// TIA Portal V17 export
// export: Created 2025-03-05T07:59:45.6753335Z, ExportSetting WithDefaults, DisplayName Totally Integrated Automation Portal, DisplayVersion V17 Update 8, DisplayName TIA Portal Openness, DisplayVersion V17 Update 8, DisplayName TIA Portal Version Control Interface, DisplayVersion V17, DisplayName SINAMICS Startdrive Advanced, DisplayVersion V17 SP2, DisplayName SINAMICS Startdrive G110M, G120, G120C, G120D, G120P, G115D, DisplayVersion V17 SP2, DisplayName SINAMICS Startdrive G130, G150, S120, S150, SINAMICS MV, S210, DisplayVersion V17 SP2, DisplayName STEP 7 Professional, DisplayVersion V17 Update 8, DisplayName SINUMERIK ONE STEP 7 Toolbox, DisplayVersion V17 Update 12, DisplayName SINUMERIK 840D sl STEP 7 Toolbox, DisplayVersion V17 Update 12, DisplayName STEP 7 Safety, DisplayVersion V17 Update 6, DisplayName WinCC Advanced, DisplayVersion V17 Update 8
FUNCTION "FC326_CHANNEL_6" : Void   // FC326, LAD
{ S7_Optimized_Access := 'FALSE' }
AUTHOR : ETXETAR
VERSION : 1.0
// stored: AutoNumber false, IsIECCheckEnabled false, SetENOAutomatically false, UDAEnableTagReadback false
   VAR_TEMP
      NC_RESET_CH2 : Bool;
      NC_START_CH2 : Bool;
   END_VAR
BEGIN

REGION Network 1: RESET CHANNEL
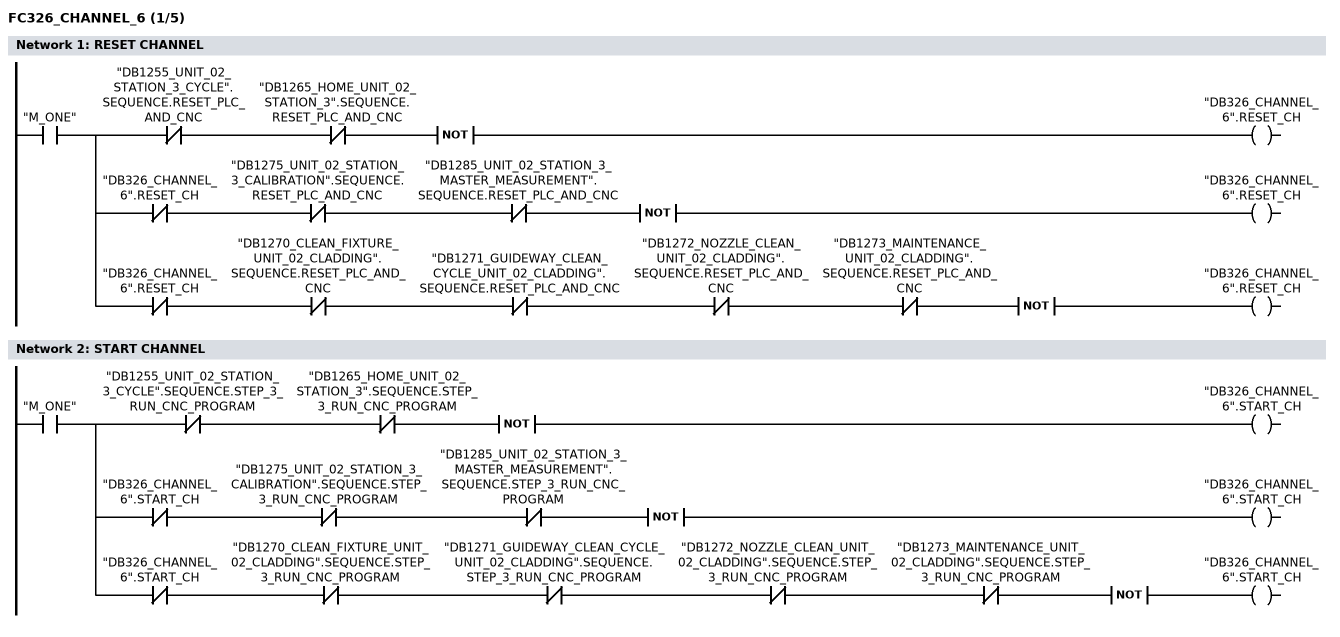
   RUNG wire#powerrail
      Contact( "M_ONE" )
      wire#w1
      I_Contact( "DB1255_UNIT_02_STATION_3_CYCLE".SEQUENCE.RESET_PLC_AND_CNC )
      I_Contact( "DB1265_HOME_UNIT_02_STATION_3".SEQUENCE.RESET_PLC_AND_CNC )
      Not()
      Coil( "DB326_CHANNEL_6".RESET_CH )
   END_RUNG
   RUNG wire#w1
      I_Contact( "DB326_CHANNEL_6".RESET_CH )
      I_Contact( "DB1275_UNIT_02_STATION_3_CALIBRATION".SEQUENCE.RESET_PLC_AND_CNC )
      I_Contact( "DB1285_UNIT_02_STATION_3_MASTER_MEASUREMENT".SEQUENCE.RESET_PLC_AND_CNC )
      Not()
      Coil( "DB326_CHANNEL_6".RESET_CH )
   END_RUNG
   RUNG wire#w1
      I_Contact( "DB326_CHANNEL_6".RESET_CH )
      I_Contact( "DB1270_CLEAN_FIXTURE_UNIT_02_CLADDING".SEQUENCE.RESET_PLC_AND_CNC )
      I_Contact( "DB1271_GUIDEWAY_CLEAN_CYCLE_UNIT_02_CLADDING".SEQUENCE.RESET_PLC_AND_CNC )
      I_Contact( "DB1272_NOZZLE_CLEAN_UNIT_02_CLADDING".SEQUENCE.RESET_PLC_AND_CNC )
      I_Contact( "DB1273_MAINTENANCE_UNIT_02_CLADDING".SEQUENCE.RESET_PLC_AND_CNC )
      Not()
      Coil( "DB326_CHANNEL_6".RESET_CH )
   END_RUNG
   // the same network as SCL:
   "DB326_CHANNEL_6".RESET_CH := NOT ("M_ONE" AND NOT "DB1255_UNIT_02_STATION_3_CYCLE".SEQUENCE.RESET_PLC_AND_CNC AND NOT "DB1265_HOME_UNIT_02_STATION_3".SEQUENCE.RESET_PLC_AND_CNC);
   "DB326_CHANNEL_6".RESET_CH := NOT ("M_ONE" AND NOT "DB326_CHANNEL_6".RESET_CH AND NOT "DB1275_UNIT_02_STATION_3_CALIBRATION".SEQUENCE.RESET_PLC_AND_CNC AND NOT "DB1285_UNIT_02_STATION_3_MASTER_MEASUREMENT".SEQUENCE.RESET_PLC_AND_CNC);
   "DB326_CHANNEL_6".RESET_CH := NOT ("M_ONE" AND NOT "DB326_CHANNEL_6".RESET_CH AND NOT "DB1270_CLEAN_FIXTURE_UNIT_02_CLADDING".SEQUENCE.RESET_PLC_AND_CNC AND NOT "DB1271_GUIDEWAY_CLEAN_CYCLE_UNIT_02_CLADDING".SEQUENCE.RESET_PLC_AND_CNC AND NOT "DB1272_NOZZLE_CLEAN_UNIT_02_CLADDING".SEQUENCE.RESET_PLC_AND_CNC AND NOT "DB1273_MAINTENANCE_UNIT_02_CLADDING".SEQUENCE.RESET_PLC_AND_CNC);
END_REGION

REGION Network 2: START CHANNEL
   RUNG wire#powerrail
      Contact( "M_ONE" )
      wire#w1
      I_Contact( "DB1255_UNIT_02_STATION_3_CYCLE".SEQUENCE.STEP_3_RUN_CNC_PROGRAM )
      I_Contact( "DB1265_HOME_UNIT_02_STATION_3".SEQUENCE.STEP_3_RUN_CNC_PROGRAM )
      Not()
      Coil( "DB326_CHANNEL_6".START_CH )
   END_RUNG
   RUNG wire#w1
      I_Contact( "DB326_CHANNEL_6".START_CH )
      I_Contact( "DB1275_UNIT_02_STATION_3_CALIBRATION".SEQUENCE.STEP_3_RUN_CNC_PROGRAM )
      I_Contact( "DB1285_UNIT_02_STATION_3_MASTER_MEASUREMENT".SEQUENCE.STEP_3_RUN_CNC_PROGRAM )
      Not()
      Coil( "DB326_CHANNEL_6".START_CH )
   END_RUNG
   RUNG wire#w1
      I_Contact( "DB326_CHANNEL_6".START_CH )
      I_Contact( "DB1270_CLEAN_FIXTURE_UNIT_02_CLADDING".SEQUENCE.STEP_3_RUN_CNC_PROGRAM )
      I_Contact( "DB1271_GUIDEWAY_CLEAN_CYCLE_UNIT_02_CLADDING".SEQUENCE.STEP_3_RUN_CNC_PROGRAM )
      I_Contact( "DB1272_NOZZLE_CLEAN_UNIT_02_CLADDING".SEQUENCE.STEP_3_RUN_CNC_PROGRAM )
      I_Contact( "DB1273_MAINTENANCE_UNIT_02_CLADDING".SEQUENCE.STEP_3_RUN_CNC_PROGRAM )
      Not()
      Coil( "DB326_CHANNEL_6".START_CH )
   END_RUNG
   // the same network as SCL:
   "DB326_CHANNEL_6".START_CH := NOT ("M_ONE" AND NOT "DB1255_UNIT_02_STATION_3_CYCLE".SEQUENCE.STEP_3_RUN_CNC_PROGRAM AND NOT "DB1265_HOME_UNIT_02_STATION_3".SEQUENCE.STEP_3_RUN_CNC_PROGRAM);
   "DB326_CHANNEL_6".START_CH := NOT ("M_ONE" AND NOT "DB326_CHANNEL_6".START_CH AND NOT "DB1275_UNIT_02_STATION_3_CALIBRATION".SEQUENCE.STEP_3_RUN_CNC_PROGRAM AND NOT "DB1285_UNIT_02_STATION_3_MASTER_MEASUREMENT".SEQUENCE.STEP_3_RUN_CNC_PROGRAM);
   "DB326_CHANNEL_6".START_CH := NOT ("M_ONE" AND NOT "DB326_CHANNEL_6".START_CH AND NOT "DB1270_CLEAN_FIXTURE_UNIT_02_CLADDING".SEQUENCE.STEP_3_RUN_CNC_PROGRAM AND NOT "DB1271_GUIDEWAY_CLEAN_CYCLE_UNIT_02_CLADDING".SEQUENCE.STEP_3_RUN_CNC_PROGRAM AND NOT "DB1272_NOZZLE_CLEAN_UNIT_02_CLADDING".SEQUENCE.STEP_3_RUN_CNC_PROGRAM AND NOT "DB1273_MAINTENANCE_UNIT_02_CLADDING".SEQUENCE.STEP_3_RUN_CNC_PROGRAM);
END_REGION

REGION Network 3: CALL FB321 CHANNEL 6 / CHANNEL 3 XFLEX-DUO
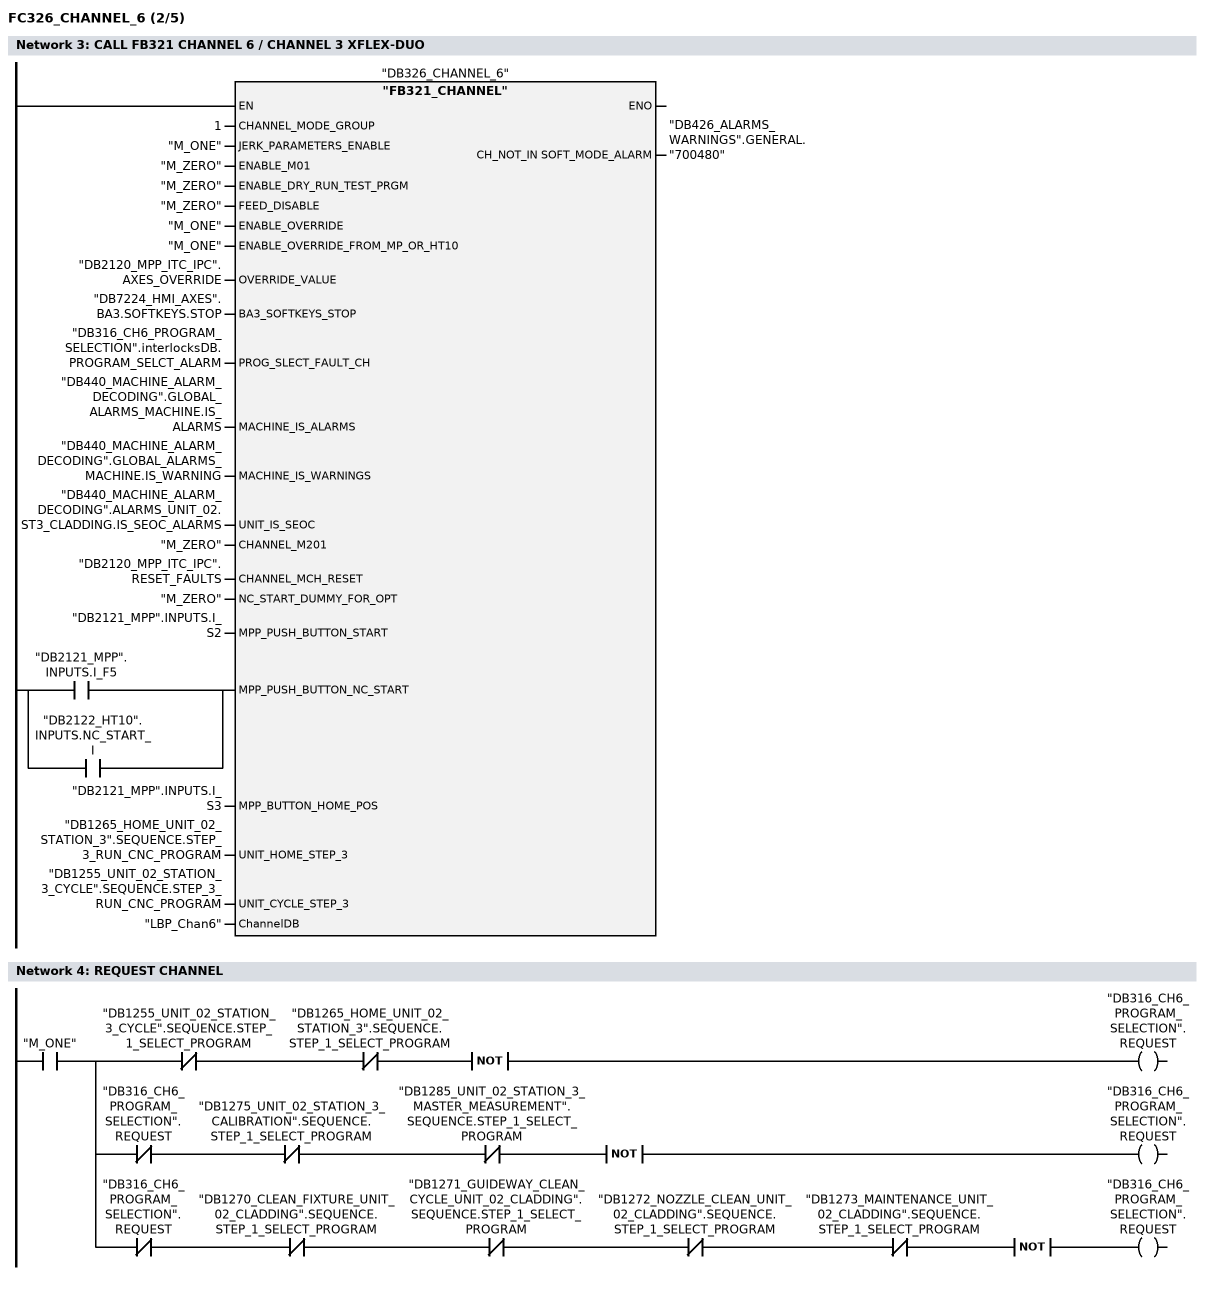
   RUNG wire#powerrail
      "DB326_CHANNEL_6"(MPP_PUSH_BUTTON_NC_START := wire#w1, CHANNEL_MODE_GROUP := 1, JERK_PARAMETERS_ENABLE := "M_ONE", ENABLE_M01 := "M_ZERO", ENABLE_DRY_RUN_TEST_PRGM := "M_ZERO", FEED_DISABLE := "M_ZERO", ENABLE_OVERRIDE := "M_ONE", ENABLE_OVERRIDE_FROM_MP_OR_HT10 := "M_ONE", OVERRIDE_VALUE := "DB2120_MPP_ITC_IPC".AXES_OVERRIDE, BA3_SOFTKEYS_STOP := "DB7224_HMI_AXES".BA3.SOFTKEYS.STOP, PROG_SLECT_FAULT_CH := "DB316_CH6_PROGRAM_SELECTION".interlocksDB.PROGRAM_SELCT_ALARM, MACHINE_IS_ALARMS := "DB440_MACHINE_ALARM_DECODING".GLOBAL_ALARMS_MACHINE.IS_ALARMS, MACHINE_IS_WARNINGS := "DB440_MACHINE_ALARM_DECODING".GLOBAL_ALARMS_MACHINE.IS_WARNING, UNIT_IS_SEOC := "DB440_MACHINE_ALARM_DECODING".ALARMS_UNIT_02.ST3_CLADDING.IS_SEOC_ALARMS, CHANNEL_M201 := "M_ZERO", CHANNEL_MCH_RESET := "DB2120_MPP_ITC_IPC".RESET_FAULTS, NC_START_DUMMY_FOR_OPT := "M_ZERO", MPP_PUSH_BUTTON_START := "DB2121_MPP".INPUTS.I_S2, MPP_BUTTON_HOME_POS := "DB2121_MPP".INPUTS.I_S3, UNIT_HOME_STEP_3 := "DB1265_HOME_UNIT_02_STATION_3".SEQUENCE.STEP_3_RUN_CNC_PROGRAM, UNIT_CYCLE_STEP_3 := "DB1255_UNIT_02_STATION_3_CYCLE".SEQUENCE.STEP_3_RUN_CNC_PROGRAM, ChannelDB := "LBP_Chan6", "CH_NOT_IN SOFT_MODE_ALARM" => "DB426_ALARMS_WARNINGS".GENERAL."700480")
   END_RUNG
   RUNG wire#powerrail
      Contact( "DB2121_MPP".INPUTS.I_F5 )
   END_RUNG wire#w1
   RUNG wire#powerrail
      Contact( "DB2122_HT10".INPUTS.NC_START_I )
   END_RUNG wire#w1
   // the same network as SCL:
   "DB326_CHANNEL_6"(CHANNEL_MODE_GROUP := 1,   // "FB321_CHANNEL"
                     JERK_PARAMETERS_ENABLE := "M_ONE",
                     ENABLE_M01 := "M_ZERO",
                     ENABLE_DRY_RUN_TEST_PRGM := "M_ZERO",
                     FEED_DISABLE := "M_ZERO",
                     ENABLE_OVERRIDE := "M_ONE",
                     ENABLE_OVERRIDE_FROM_MP_OR_HT10 := "M_ONE",
                     OVERRIDE_VALUE := "DB2120_MPP_ITC_IPC".AXES_OVERRIDE,
                     BA3_SOFTKEYS_STOP := "DB7224_HMI_AXES".BA3.SOFTKEYS.STOP,
                     PROG_SLECT_FAULT_CH := "DB316_CH6_PROGRAM_SELECTION".interlocksDB.PROGRAM_SELCT_ALARM,
                     MACHINE_IS_ALARMS := "DB440_MACHINE_ALARM_DECODING".GLOBAL_ALARMS_MACHINE.IS_ALARMS,
                     MACHINE_IS_WARNINGS := "DB440_MACHINE_ALARM_DECODING".GLOBAL_ALARMS_MACHINE.IS_WARNING,
                     UNIT_IS_SEOC := "DB440_MACHINE_ALARM_DECODING".ALARMS_UNIT_02.ST3_CLADDING.IS_SEOC_ALARMS,
                     CHANNEL_M201 := "M_ZERO",
                     CHANNEL_MCH_RESET := "DB2120_MPP_ITC_IPC".RESET_FAULTS,
                     NC_START_DUMMY_FOR_OPT := "M_ZERO",
                     MPP_PUSH_BUTTON_START := "DB2121_MPP".INPUTS.I_S2,
                     MPP_PUSH_BUTTON_NC_START := "DB2121_MPP".INPUTS.I_F5 OR "DB2122_HT10".INPUTS.NC_START_I,
                     MPP_BUTTON_HOME_POS := "DB2121_MPP".INPUTS.I_S3,
                     UNIT_HOME_STEP_3 := "DB1265_HOME_UNIT_02_STATION_3".SEQUENCE.STEP_3_RUN_CNC_PROGRAM,
                     UNIT_CYCLE_STEP_3 := "DB1255_UNIT_02_STATION_3_CYCLE".SEQUENCE.STEP_3_RUN_CNC_PROGRAM,
                     ChannelDB := "LBP_Chan6",
                     "CH_NOT_IN SOFT_MODE_ALARM" => "DB426_ALARMS_WARNINGS".GENERAL."700480");
END_REGION

REGION Network 4: REQUEST CHANNEL
   RUNG wire#powerrail
      Contact( "M_ONE" )
      wire#w1
      I_Contact( "DB1255_UNIT_02_STATION_3_CYCLE".SEQUENCE.STEP_1_SELECT_PROGRAM )
      I_Contact( "DB1265_HOME_UNIT_02_STATION_3".SEQUENCE.STEP_1_SELECT_PROGRAM )
      Not()
      Coil( "DB316_CH6_PROGRAM_SELECTION".REQUEST )
   END_RUNG
   RUNG wire#w1
      I_Contact( "DB316_CH6_PROGRAM_SELECTION".REQUEST )
      I_Contact( "DB1275_UNIT_02_STATION_3_CALIBRATION".SEQUENCE.STEP_1_SELECT_PROGRAM )
      I_Contact( "DB1285_UNIT_02_STATION_3_MASTER_MEASUREMENT".SEQUENCE.STEP_1_SELECT_PROGRAM )
      Not()
      Coil( "DB316_CH6_PROGRAM_SELECTION".REQUEST )
   END_RUNG
   RUNG wire#w1
      I_Contact( "DB316_CH6_PROGRAM_SELECTION".REQUEST )
      I_Contact( "DB1270_CLEAN_FIXTURE_UNIT_02_CLADDING".SEQUENCE.STEP_1_SELECT_PROGRAM )
      I_Contact( "DB1271_GUIDEWAY_CLEAN_CYCLE_UNIT_02_CLADDING".SEQUENCE.STEP_1_SELECT_PROGRAM )
      I_Contact( "DB1272_NOZZLE_CLEAN_UNIT_02_CLADDING".SEQUENCE.STEP_1_SELECT_PROGRAM )
      I_Contact( "DB1273_MAINTENANCE_UNIT_02_CLADDING".SEQUENCE.STEP_1_SELECT_PROGRAM )
      Not()
      Coil( "DB316_CH6_PROGRAM_SELECTION".REQUEST )
   END_RUNG
   // the same network as SCL:
   "DB316_CH6_PROGRAM_SELECTION".REQUEST := NOT ("M_ONE" AND NOT "DB1255_UNIT_02_STATION_3_CYCLE".SEQUENCE.STEP_1_SELECT_PROGRAM AND NOT "DB1265_HOME_UNIT_02_STATION_3".SEQUENCE.STEP_1_SELECT_PROGRAM);
   "DB316_CH6_PROGRAM_SELECTION".REQUEST := NOT ("M_ONE" AND NOT "DB316_CH6_PROGRAM_SELECTION".REQUEST AND NOT "DB1275_UNIT_02_STATION_3_CALIBRATION".SEQUENCE.STEP_1_SELECT_PROGRAM AND NOT "DB1285_UNIT_02_STATION_3_MASTER_MEASUREMENT".SEQUENCE.STEP_1_SELECT_PROGRAM);
   "DB316_CH6_PROGRAM_SELECTION".REQUEST := NOT ("M_ONE" AND NOT "DB316_CH6_PROGRAM_SELECTION".REQUEST AND NOT "DB1270_CLEAN_FIXTURE_UNIT_02_CLADDING".SEQUENCE.STEP_1_SELECT_PROGRAM AND NOT "DB1271_GUIDEWAY_CLEAN_CYCLE_UNIT_02_CLADDING".SEQUENCE.STEP_1_SELECT_PROGRAM AND NOT "DB1272_NOZZLE_CLEAN_UNIT_02_CLADDING".SEQUENCE.STEP_1_SELECT_PROGRAM AND NOT "DB1273_MAINTENANCE_UNIT_02_CLADDING".SEQUENCE.STEP_1_SELECT_PROGRAM);
END_REGION

REGION Network 5: CALL FB311 CHANNEL PROGRAM SELECTION / CHANNEL 3 X-FLEX DUO
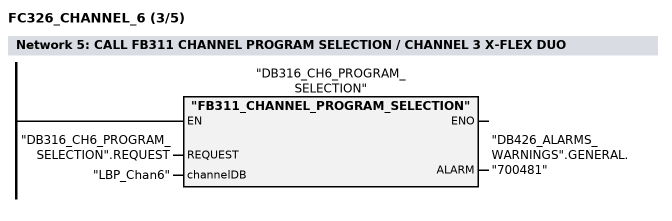
   RUNG wire#powerrail
      "DB316_CH6_PROGRAM_SELECTION"(REQUEST := "DB316_CH6_PROGRAM_SELECTION".REQUEST, channelDB := "LBP_Chan6", ALARM => "DB426_ALARMS_WARNINGS".GENERAL."700481")
   END_RUNG
   // the same network as SCL:
   "DB316_CH6_PROGRAM_SELECTION"(REQUEST := "DB316_CH6_PROGRAM_SELECTION".REQUEST,   // "FB311_CHANNEL_PROGRAM_SELECTION"
                           channelDB := "LBP_Chan6",
                           ALARM => "DB426_ALARMS_WARNINGS".GENERAL."700481");
END_REGION

REGION Network 6: CALL FB301 CHANNEL READ AXES POSITIONS
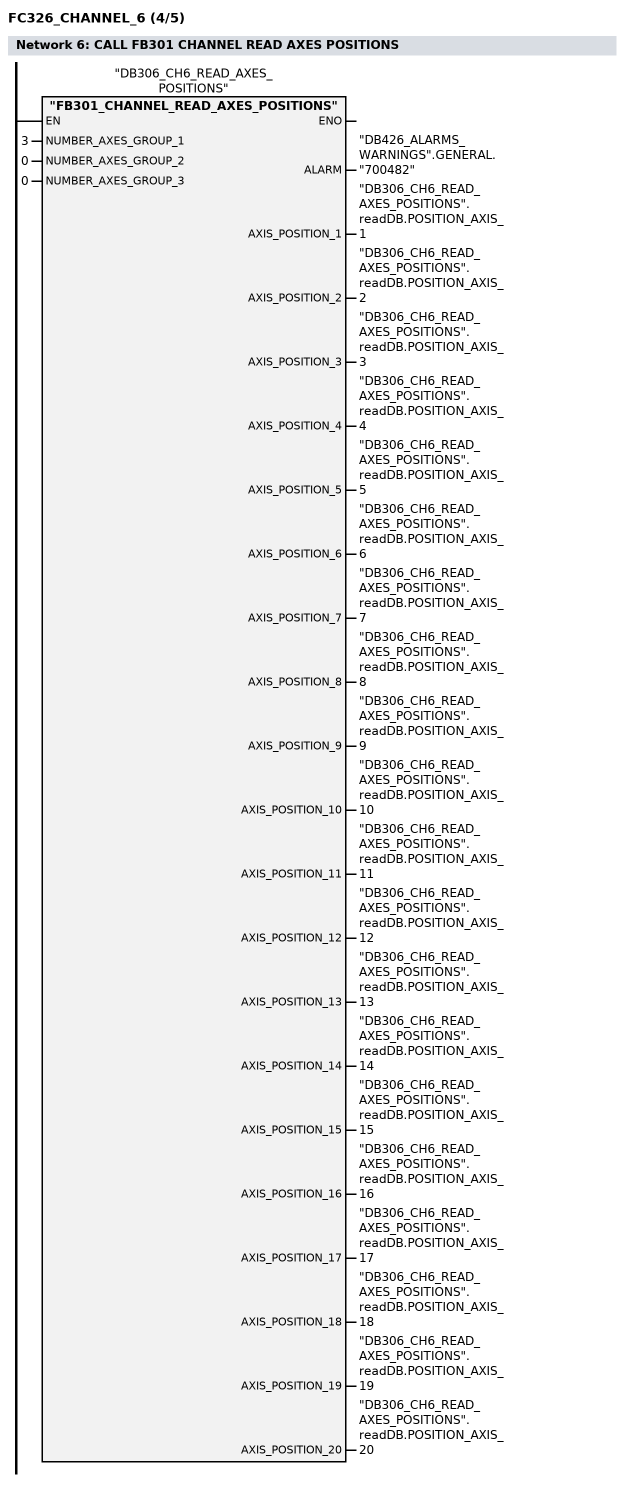
   RUNG wire#powerrail
      "DB306_CH6_READ_AXES_POSITIONS"(NUMBER_AXES_GROUP_1 := 3, NUMBER_AXES_GROUP_2 := 0, NUMBER_AXES_GROUP_3 := 0, ALARM => "DB426_ALARMS_WARNINGS".GENERAL."700482", AXIS_POSITION_1 => "DB306_CH6_READ_AXES_POSITIONS".readDB.POSITION_AXIS_1, AXIS_POSITION_2 => "DB306_CH6_READ_AXES_POSITIONS".readDB.POSITION_AXIS_2, AXIS_POSITION_3 => "DB306_CH6_READ_AXES_POSITIONS".readDB.POSITION_AXIS_3, AXIS_POSITION_4 => "DB306_CH6_READ_AXES_POSITIONS".readDB.POSITION_AXIS_4, AXIS_POSITION_5 => "DB306_CH6_READ_AXES_POSITIONS".readDB.POSITION_AXIS_5, AXIS_POSITION_6 => "DB306_CH6_READ_AXES_POSITIONS".readDB.POSITION_AXIS_6, AXIS_POSITION_7 => "DB306_CH6_READ_AXES_POSITIONS".readDB.POSITION_AXIS_7, AXIS_POSITION_8 => "DB306_CH6_READ_AXES_POSITIONS".readDB.POSITION_AXIS_8, AXIS_POSITION_9 => "DB306_CH6_READ_AXES_POSITIONS".readDB.POSITION_AXIS_9, AXIS_POSITION_10 => "DB306_CH6_READ_AXES_POSITIONS".readDB.POSITION_AXIS_10, AXIS_POSITION_11 => "DB306_CH6_READ_AXES_POSITIONS".readDB.POSITION_AXIS_11, AXIS_POSITION_12 => "DB306_CH6_READ_AXES_POSITIONS".readDB.POSITION_AXIS_12, AXIS_POSITION_13 => "DB306_CH6_READ_AXES_POSITIONS".readDB.POSITION_AXIS_13, AXIS_POSITION_14 => "DB306_CH6_READ_AXES_POSITIONS".readDB.POSITION_AXIS_14, AXIS_POSITION_15 => "DB306_CH6_READ_AXES_POSITIONS".readDB.POSITION_AXIS_15, AXIS_POSITION_16 => "DB306_CH6_READ_AXES_POSITIONS".readDB.POSITION_AXIS_16, AXIS_POSITION_17 => "DB306_CH6_READ_AXES_POSITIONS".readDB.POSITION_AXIS_17, AXIS_POSITION_18 => "DB306_CH6_READ_AXES_POSITIONS".readDB.POSITION_AXIS_18, AXIS_POSITION_19 => "DB306_CH6_READ_AXES_POSITIONS".readDB.POSITION_AXIS_19, AXIS_POSITION_20 => "DB306_CH6_READ_AXES_POSITIONS".readDB.POSITION_AXIS_20)
   END_RUNG
   // the same network as SCL:
   "DB306_CH6_READ_AXES_POSITIONS"(NUMBER_AXES_GROUP_1 := 3,   // "FB301_CHANNEL_READ_AXES_POSITIONS"
                           NUMBER_AXES_GROUP_2 := 0,
                           NUMBER_AXES_GROUP_3 := 0,
                           ALARM => "DB426_ALARMS_WARNINGS".GENERAL."700482",
                           AXIS_POSITION_1 => "DB306_CH6_READ_AXES_POSITIONS".readDB.POSITION_AXIS_1,
                           AXIS_POSITION_2 => "DB306_CH6_READ_AXES_POSITIONS".readDB.POSITION_AXIS_2,
                           AXIS_POSITION_3 => "DB306_CH6_READ_AXES_POSITIONS".readDB.POSITION_AXIS_3,
                           AXIS_POSITION_4 => "DB306_CH6_READ_AXES_POSITIONS".readDB.POSITION_AXIS_4,
                           AXIS_POSITION_5 => "DB306_CH6_READ_AXES_POSITIONS".readDB.POSITION_AXIS_5,
                           AXIS_POSITION_6 => "DB306_CH6_READ_AXES_POSITIONS".readDB.POSITION_AXIS_6,
                           AXIS_POSITION_7 => "DB306_CH6_READ_AXES_POSITIONS".readDB.POSITION_AXIS_7,
                           AXIS_POSITION_8 => "DB306_CH6_READ_AXES_POSITIONS".readDB.POSITION_AXIS_8,
                           AXIS_POSITION_9 => "DB306_CH6_READ_AXES_POSITIONS".readDB.POSITION_AXIS_9,
                           AXIS_POSITION_10 => "DB306_CH6_READ_AXES_POSITIONS".readDB.POSITION_AXIS_10,
                           AXIS_POSITION_11 => "DB306_CH6_READ_AXES_POSITIONS".readDB.POSITION_AXIS_11,
                           AXIS_POSITION_12 => "DB306_CH6_READ_AXES_POSITIONS".readDB.POSITION_AXIS_12,
                           AXIS_POSITION_13 => "DB306_CH6_READ_AXES_POSITIONS".readDB.POSITION_AXIS_13,
                           AXIS_POSITION_14 => "DB306_CH6_READ_AXES_POSITIONS".readDB.POSITION_AXIS_14,
                           AXIS_POSITION_15 => "DB306_CH6_READ_AXES_POSITIONS".readDB.POSITION_AXIS_15,
                           AXIS_POSITION_16 => "DB306_CH6_READ_AXES_POSITIONS".readDB.POSITION_AXIS_16,
                           AXIS_POSITION_17 => "DB306_CH6_READ_AXES_POSITIONS".readDB.POSITION_AXIS_17,
                           AXIS_POSITION_18 => "DB306_CH6_READ_AXES_POSITIONS".readDB.POSITION_AXIS_18,
                           AXIS_POSITION_19 => "DB306_CH6_READ_AXES_POSITIONS".readDB.POSITION_AXIS_19,
                           AXIS_POSITION_20 => "DB306_CH6_READ_AXES_POSITIONS".readDB.POSITION_AXIS_20);
END_REGION

REGION Network 7: CALL FC341 NCK M STA 3 / CALL FC1181
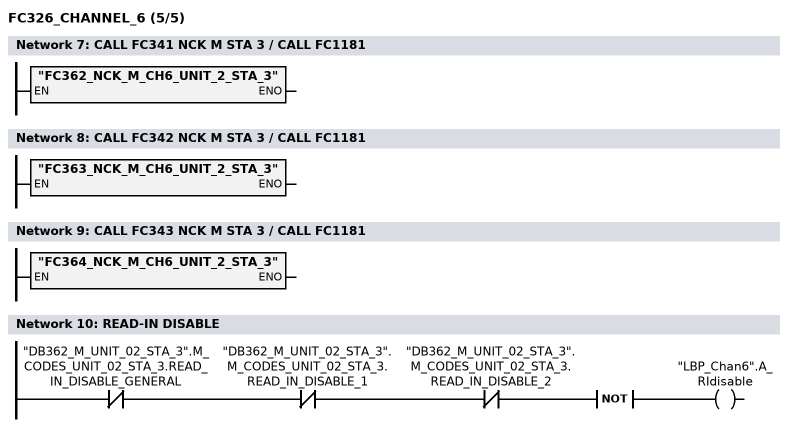
   RUNG wire#powerrail
      "FC362_NCK_M_CH6_UNIT_2_STA_3"()
   END_RUNG
   // the same network as SCL:
   "FC362_NCK_M_CH6_UNIT_2_STA_3"();
END_REGION

REGION Network 8: CALL FC342 NCK M STA 3 / CALL FC1181
   RUNG wire#powerrail
      "FC363_NCK_M_CH6_UNIT_2_STA_3"()
   END_RUNG
   // the same network as SCL:
   "FC363_NCK_M_CH6_UNIT_2_STA_3"();
END_REGION

REGION Network 9: CALL FC343 NCK M STA 3 / CALL FC1181
   RUNG wire#powerrail
      "FC364_NCK_M_CH6_UNIT_2_STA_3"()
   END_RUNG
   // the same network as SCL:
   "FC364_NCK_M_CH6_UNIT_2_STA_3"();
END_REGION

REGION Network 10: READ-IN DISABLE
   RUNG wire#powerrail
      I_Contact( "DB362_M_UNIT_02_STA_3".M_CODES_UNIT_02_STA_3.READ_IN_DISABLE_GENERAL )
      I_Contact( "DB362_M_UNIT_02_STA_3".M_CODES_UNIT_02_STA_3.READ_IN_DISABLE_1 )
      I_Contact( "DB362_M_UNIT_02_STA_3".M_CODES_UNIT_02_STA_3.READ_IN_DISABLE_2 )
      Not()
      Coil( "LBP_Chan6".A_RIdisable )
   END_RUNG
   // the same network as SCL:
   "LBP_Chan6".A_RIdisable := NOT (NOT "DB362_M_UNIT_02_STA_3".M_CODES_UNIT_02_STA_3.READ_IN_DISABLE_GENERAL AND NOT "DB362_M_UNIT_02_STA_3".M_CODES_UNIT_02_STA_3.READ_IN_DISABLE_1 AND NOT "DB362_M_UNIT_02_STA_3".M_CODES_UNIT_02_STA_3.READ_IN_DISABLE_2);
END_REGION
END_FUNCTION
